TYPE ST_ToVisuSensorActor :
STRUCT
	stType			: ST_Text;
	stName			: ST_Text;
	stBMK			: ST_Text;
	stZustand		: ST_Text;
END_STRUCT
END_TYPE

(* stored: Version 1.1.0.1, ProductVersion 3.1.4024.11
   DUT ST_ToVisuSensorActor: Id {bd02fdf0-6d3e-4c55-afe7-8b3c322470fe} *)
